(* Logix 5000 project; controller cal1632 1756-L62 rev 16.20; software revision 16.05; part 49 of 61 *)
(* tags used below, declared in another part *)
   FAULT : BOOL;
   HMI : BOOL;
   p01_recipe_active : recipe;
   p01r02 : routine;
   p01r09_pb_global_reset : BOOL;
   p27_ao_dia_a : REAL;
   p27_ao_dia_b : REAL;
   p27_inactive_tension_sp : REAL;
   p27r03_lower_A_tension_on : BOOL;
   p27r03_lower_B_tension_on : BOOL;
   p27r10 : routine;
   p27r10_lla_selected_tension : REAL;
   p27r10_llb_selected_tension : REAL;
   p27r10_timer_fault : TIMER[4];
   p27r10_timer_warning : TIMER[4];
   p27r10_unwind_a_brake_torque : REAL;
   p27r10_unwind_a_dia_ft : REAL;
   p27r10_unwind_b_brake_torque : REAL;
   p27r10_unwind_b_dia_ft : REAL;
   p28_ai_slitter_amps : REAL;
   p28_ai_slitter_hz : REAL;
   p28_ai_slitter_speed : REAL;
   p28_ao_sltr_selected_speed : REAL;
   p28_di_brake : BOOL;
   p28_di_motor : BOOL;
   p28_di_slitter : acs800_di_normal;
   p28_dint_to_hmi : DINT[16];
   p28_do_slt_air_supply_sv : BOOL;
   p28_do_sltr : acs800_do_normal;
   p28r01 : routine;
   p28r02 : routine;
   p28r02_fault_exists : BOOL;
   p28r02_timer_fault : TIMER[4];
   p28r02_timer_warning : TIMER[4];
   p28r02_unack_fault : BOOL;
   p28r02_unack_warning : BOOL;
   p28r02_warning_exists : BOOL;
   p28r03 : routine;
   p28r03_hz : SYS_SCP;
   p28r03_slitter_speed_fb : SYS_RPM_TO_SPEED;
   p28r03_timer_fault : TIMER[4];
   p28r03_timer_warning : TIMER[4];
   p28r04 : routine;
   p28r04_slitter_gear_ratio : REAL;
   p28r04_slitter_roll_diameter_ft : REAL;
   p28r04_slitter_speed : SYS_SPEED_TO_VFD;
   p28r04_timer_fault : TIMER[4];
   p28r04_timer_warning : TIMER[4];
   p28r05 : routine;
   p28r05_timer_fault : TIMER[4];
   p28r05_timer_warning : TIMER[4];
   p28r06 : routine;
   p28r07 : routine;
   p28r08 : routine;
   p28r09 : routine;
   p28r10_request_line_run : BOOL;
   p28r11 : routine;
   p28r11_slitter_on : BOOL;
(* P27_Lower_Poly_Letoff, continued *)

ROUTINE R10_Tension   (* ladder *)
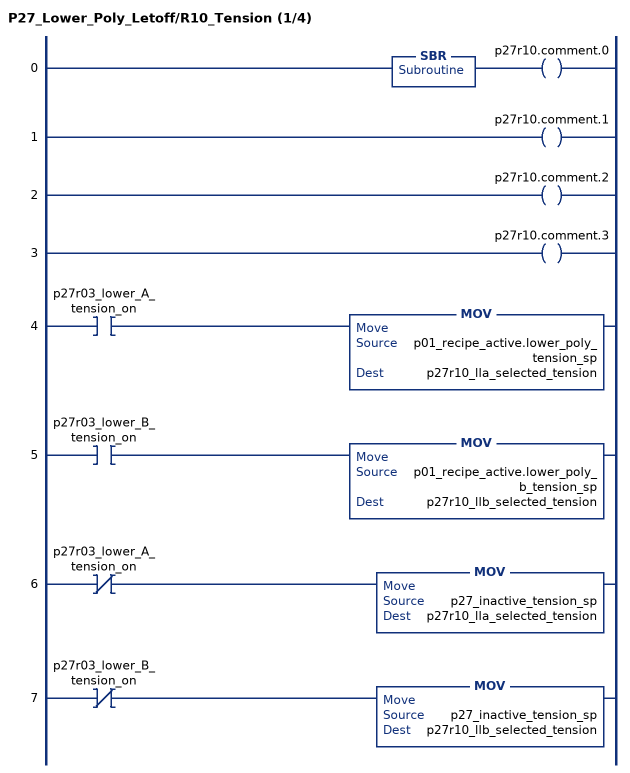
   0: SBR()OTE(p27r10.comment.0);
   1: OTE(p27r10.comment.1);
   2: OTE(p27r10.comment.2);
   3: OTE(p27r10.comment.3);
   4: XIC(p27r03_lower_A_tension_on)MOV(p01_recipe_active.lower_poly_tension_sp,p27r10_lla_selected_tension);
   5: XIC(p27r03_lower_B_tension_on)MOV(p01_recipe_active.lower_poly_b_tension_sp,p27r10_llb_selected_tension);
   6: XIO(p27r03_lower_A_tension_on)MOV(p27_inactive_tension_sp,p27r10_lla_selected_tension);
   7: XIO(p27r03_lower_B_tension_on)MOV(p27_inactive_tension_sp,p27r10_llb_selected_tension);
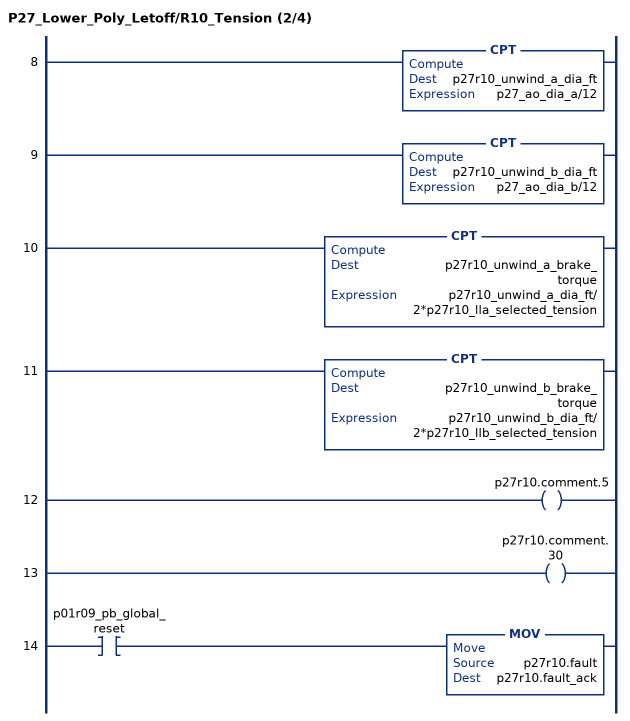
   8: CPT(p27r10_unwind_a_dia_ft,p27_ao_dia_a/12);
   9: CPT(p27r10_unwind_b_dia_ft,p27_ao_dia_b/12);
   10: CPT(p27r10_unwind_a_brake_torque,p27r10_unwind_a_dia_ft/2*p27r10_lla_selected_tension);
   11: CPT(p27r10_unwind_b_brake_torque,p27r10_unwind_b_dia_ft/2*p27r10_llb_selected_tension);
   12: OTE(p27r10.comment.5);
   13: OTE(p27r10.comment.30);
   14: XIC(p01r09_pb_global_reset)MOV(p27r10.fault,p27r10.fault_ack);
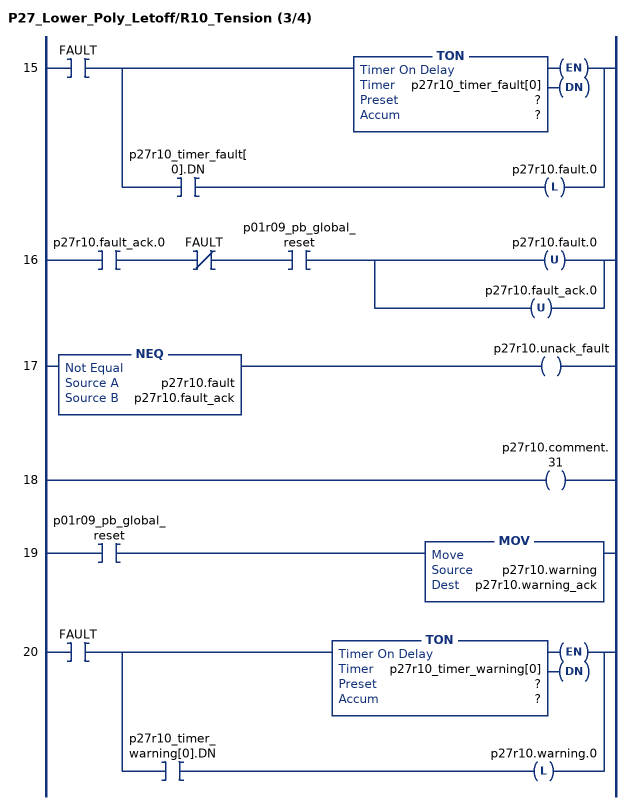
   15: XIC(FAULT)[TON(p27r10_timer_fault[0],?,?) ,XIC(p27r10_timer_fault[0].DN) OTL(p27r10.fault.0) ];
   16: XIC(p27r10.fault_ack.0)XIO(FAULT)XIC(p01r09_pb_global_reset)[OTU(p27r10.fault.0) ,OTU(p27r10.fault_ack.0) ];
   17: NEQ(p27r10.fault,p27r10.fault_ack)OTE(p27r10.unack_fault);
   18: OTE(p27r10.comment.31);
   19: XIC(p01r09_pb_global_reset)MOV(p27r10.warning,p27r10.warning_ack);
   20: XIC(FAULT)[TON(p27r10_timer_warning[0],?,?) ,XIC(p27r10_timer_warning[0].DN) OTL(p27r10.warning.0) ];
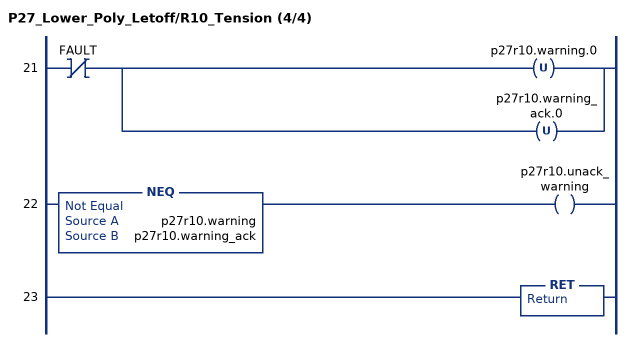
   21: XIO(FAULT)[OTU(p27r10.warning.0) ,OTU(p27r10.warning_ack.0) ];
   22: NEQ(p27r10.warning,p27r10.warning_ack)OTE(p27r10.unack_warning);
   23: RET();
END_ROUTINE
END_PROGRAM

PROGRAM P28_Slitter   (* main routine R01_Main *)

ROUTINE R01_Main   (* ladder *)
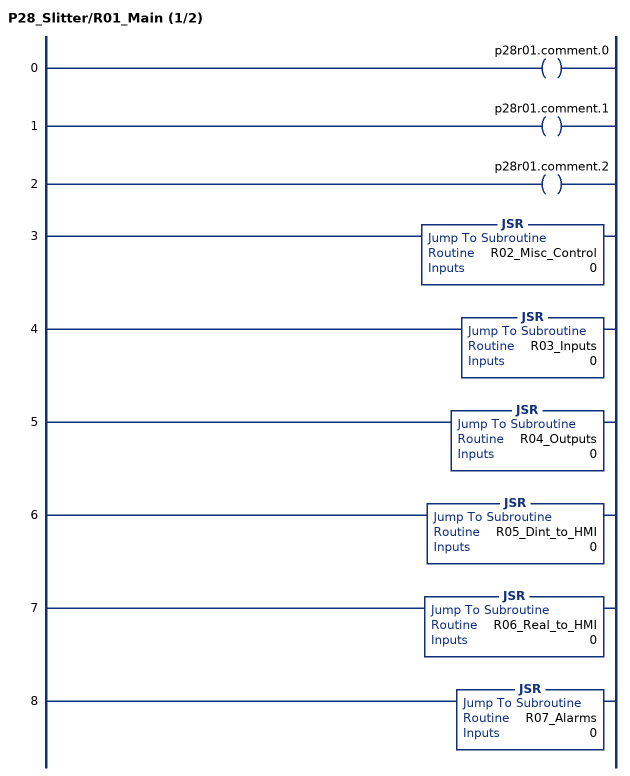
   0: OTE(p28r01.comment.0);
   1: OTE(p28r01.comment.1);
   2: OTE(p28r01.comment.2);
   3: JSR(R02_Misc_Control,0);
   4: JSR(R03_Inputs,0);
   5: JSR(R04_Outputs,0);
   6: JSR(R05_Dint_to_HMI,0);
   7: JSR(R06_Real_to_HMI,0);
   8: JSR(R07_Alarms,0);
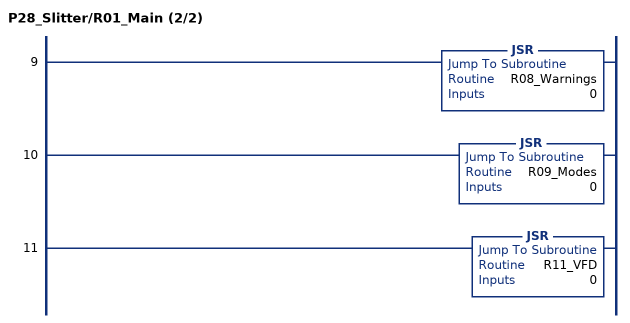
   9: JSR(R08_Warnings,0);
   10: JSR(R09_Modes,0);
   11: JSR(R11_VFD,0);
END_ROUTINE

ROUTINE R02_Misc_Control   (* ladder *)
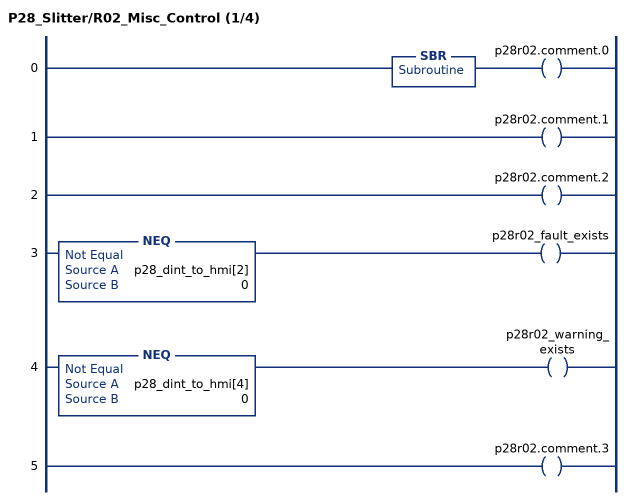
   0: SBR()OTE(p28r02.comment.0);
   1: OTE(p28r02.comment.1);
   2: OTE(p28r02.comment.2);
   3: NEQ(p28_dint_to_hmi[2],0)OTE(p28r02_fault_exists);
   4: NEQ(p28_dint_to_hmi[4],0)OTE(p28r02_warning_exists);
   5: OTE(p28r02.comment.3);
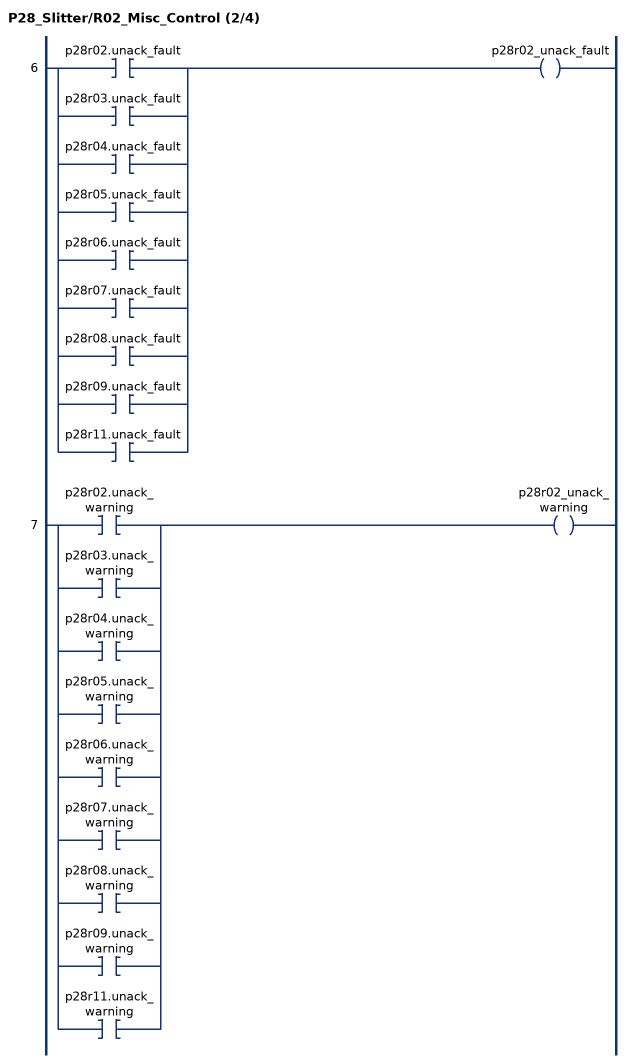
   6: [XIC(p28r02.unack_fault) ,XIC(p28r03.unack_fault) ,XIC(p28r04.unack_fault) ,XIC(p28r05.unack_fault) ,XIC(p28r06.unack_fault) ,XIC(p28r07.unack_fault) ,XIC(p28r08.unack_fault) ,XIC(p28r09.unack_fault) ,XIC(p28r11.unack_fault) ]OTE(p28r02_unack_fault);
   7: [XIC(p28r02.unack_warning) ,XIC(p28r03.unack_warning) ,XIC(p28r04.unack_warning) ,XIC(p28r05.unack_warning) ,XIC(p28r06.unack_warning) ,XIC(p28r07.unack_warning) ,XIC(p28r08.unack_warning) ,XIC(p28r09.unack_warning) ,XIC(p28r11.unack_warning) ]OTE(p28r02_unack_warning);
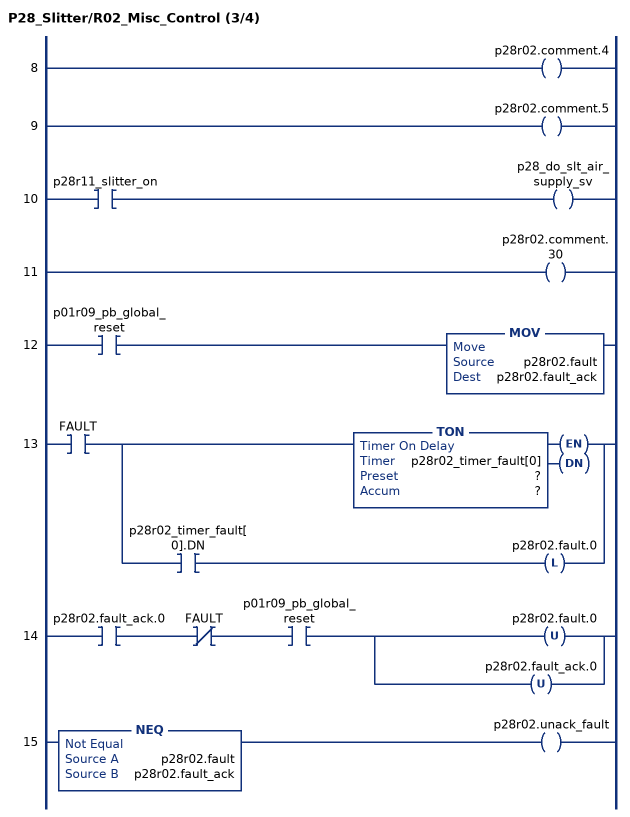
   8: OTE(p28r02.comment.4);
   9: OTE(p28r02.comment.5);
   10: XIC(p28r11_slitter_on)OTE(p28_do_slt_air_supply_sv);
   11: OTE(p28r02.comment.30);
   12: XIC(p01r09_pb_global_reset)MOV(p28r02.fault,p28r02.fault_ack);
   13: XIC(FAULT)[TON(p28r02_timer_fault[0],?,?) ,XIC(p28r02_timer_fault[0].DN) OTL(p28r02.fault.0) ];
   14: XIC(p28r02.fault_ack.0)XIO(FAULT)XIC(p01r09_pb_global_reset)[OTU(p28r02.fault.0) ,OTU(p28r02.fault_ack.0) ];
   15: NEQ(p28r02.fault,p28r02.fault_ack)OTE(p28r02.unack_fault);
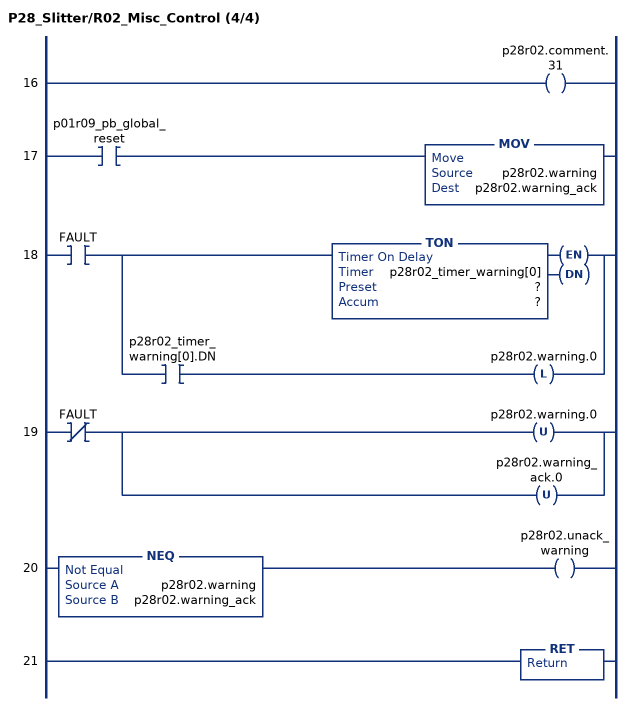
   16: OTE(p28r02.comment.31);
   17: XIC(p01r09_pb_global_reset)MOV(p28r02.warning,p28r02.warning_ack);
   18: XIC(FAULT)[TON(p28r02_timer_warning[0],?,?) ,XIC(p28r02_timer_warning[0].DN) OTL(p28r02.warning.0) ];
   19: XIO(FAULT)[OTU(p28r02.warning.0) ,OTU(p28r02.warning_ack.0) ];
   20: NEQ(p28r02.warning,p28r02.warning_ack)OTE(p28r02.unack_warning);
   21: RET();
END_ROUTINE

ROUTINE R03_Inputs   (* ladder *)
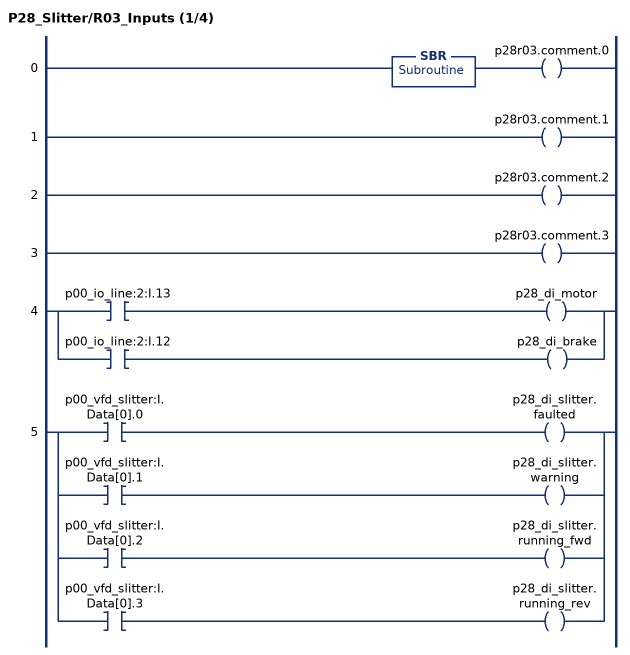
   0: SBR()OTE(p28r03.comment.0);
   1: OTE(p28r03.comment.1);
   2: OTE(p28r03.comment.2);
   3: OTE(p28r03.comment.3);
   4: [XIC(p00_io_line:2:I.13) OTE(p28_di_motor) ,XIC(p00_io_line:2:I.12) OTE(p28_di_brake) ];
   5: [XIC(p00_vfd_slitter:I.Data[0].0) OTE(p28_di_slitter.faulted) ,XIC(p00_vfd_slitter:I.Data[0].1) OTE(p28_di_slitter.warning) ,XIC(p00_vfd_slitter:I.Data[0].2) OTE(p28_di_slitter.running_fwd) ,XIC(p00_vfd_slitter:I.Data[0].3) OTE(p28_di_slitter.running_rev) ];
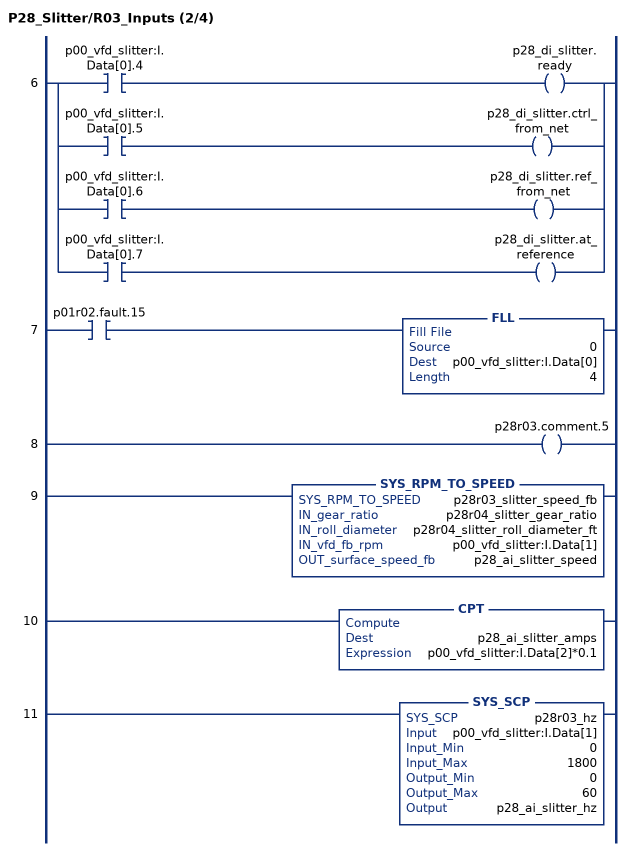
   6: [XIC(p00_vfd_slitter:I.Data[0].4) OTE(p28_di_slitter.ready) ,XIC(p00_vfd_slitter:I.Data[0].5) OTE(p28_di_slitter.ctrl_from_net) ,XIC(p00_vfd_slitter:I.Data[0].6) OTE(p28_di_slitter.ref_from_net) ,XIC(p00_vfd_slitter:I.Data[0].7) OTE(p28_di_slitter.at_reference) ];
   7: XIC(p01r02.fault.15)FLL(0,p00_vfd_slitter:I.Data[0],4);
   8: OTE(p28r03.comment.5);
   9: SYS_RPM_TO_SPEED(p28r03_slitter_speed_fb,p28r04_slitter_gear_ratio,p28r04_slitter_roll_diameter_ft,p00_vfd_slitter:I.Data[1],p28_ai_slitter_speed);
   10: CPT(p28_ai_slitter_amps,p00_vfd_slitter:I.Data[2]*0.1);
   11: SYS_SCP(p28r03_hz,p00_vfd_slitter:I.Data[1],0,1800,0,60,p28_ai_slitter_hz);
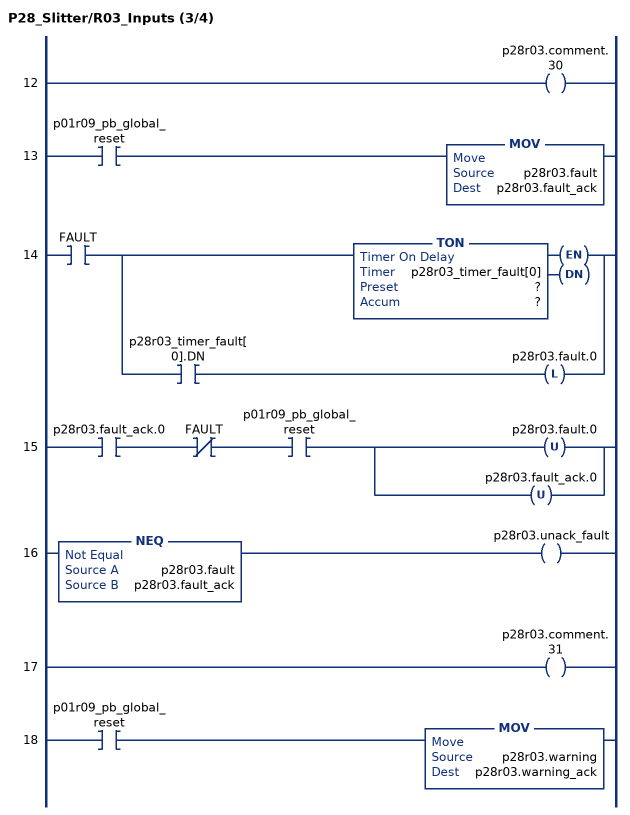
   12: OTE(p28r03.comment.30);
   13: XIC(p01r09_pb_global_reset)MOV(p28r03.fault,p28r03.fault_ack);
   14: XIC(FAULT)[TON(p28r03_timer_fault[0],?,?) ,XIC(p28r03_timer_fault[0].DN) OTL(p28r03.fault.0) ];
   15: XIC(p28r03.fault_ack.0)XIO(FAULT)XIC(p01r09_pb_global_reset)[OTU(p28r03.fault.0) ,OTU(p28r03.fault_ack.0) ];
   16: NEQ(p28r03.fault,p28r03.fault_ack)OTE(p28r03.unack_fault);
   17: OTE(p28r03.comment.31);
   18: XIC(p01r09_pb_global_reset)MOV(p28r03.warning,p28r03.warning_ack);
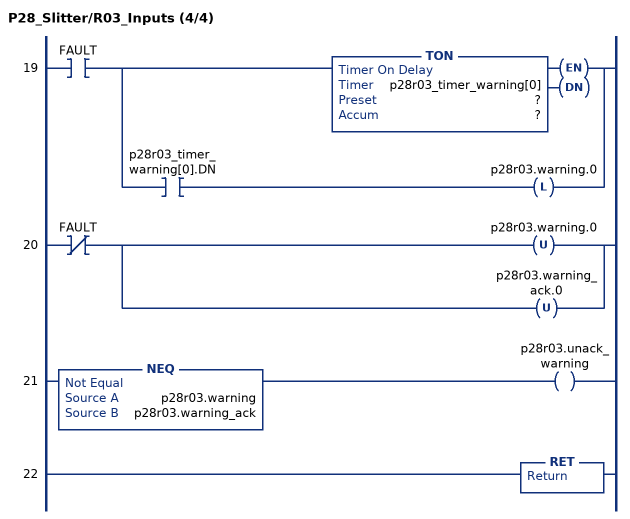
   19: XIC(FAULT)[TON(p28r03_timer_warning[0],?,?) ,XIC(p28r03_timer_warning[0].DN) OTL(p28r03.warning.0) ];
   20: XIO(FAULT)[OTU(p28r03.warning.0) ,OTU(p28r03.warning_ack.0) ];
   21: NEQ(p28r03.warning,p28r03.warning_ack)OTE(p28r03.unack_warning);
   22: RET();
END_ROUTINE

ROUTINE R04_Outputs   (* ladder *)
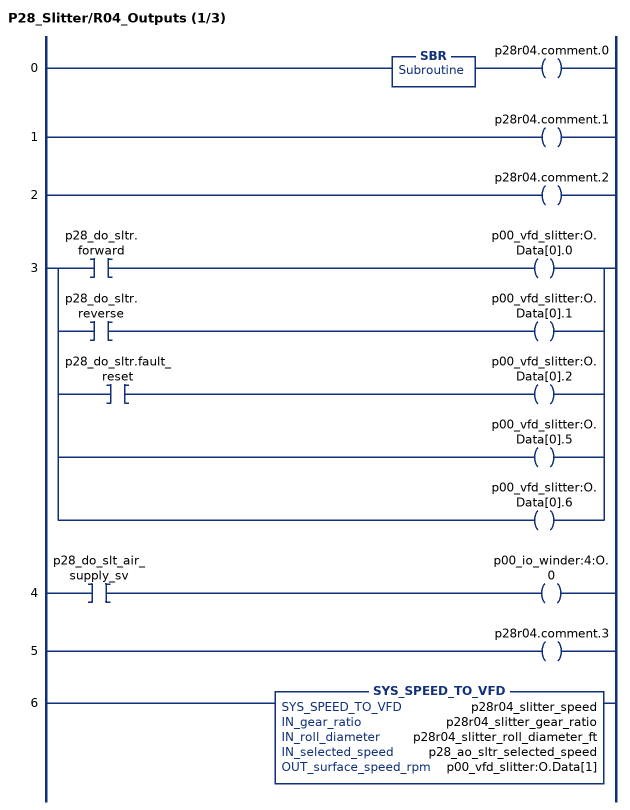
   0: SBR()OTE(p28r04.comment.0);
   1: OTE(p28r04.comment.1);
   2: OTE(p28r04.comment.2);
   3: [XIC(p28_do_sltr.forward) OTE(p00_vfd_slitter:O.Data[0].0) ,XIC(p28_do_sltr.reverse) OTE(p00_vfd_slitter:O.Data[0].1) ,XIC(p28_do_sltr.fault_reset) OTE(p00_vfd_slitter:O.Data[0].2) ,OTE(p00_vfd_slitter:O.Data[0].5) ,OTE(p00_vfd_slitter:O.Data[0].6) ];
   4: XIC(p28_do_slt_air_supply_sv)OTE(p00_io_winder:4:O.0);
   5: OTE(p28r04.comment.3);
   6: SYS_SPEED_TO_VFD(p28r04_slitter_speed,p28r04_slitter_gear_ratio,p28r04_slitter_roll_diameter_ft,p28_ao_sltr_selected_speed,p00_vfd_slitter:O.Data[1]);
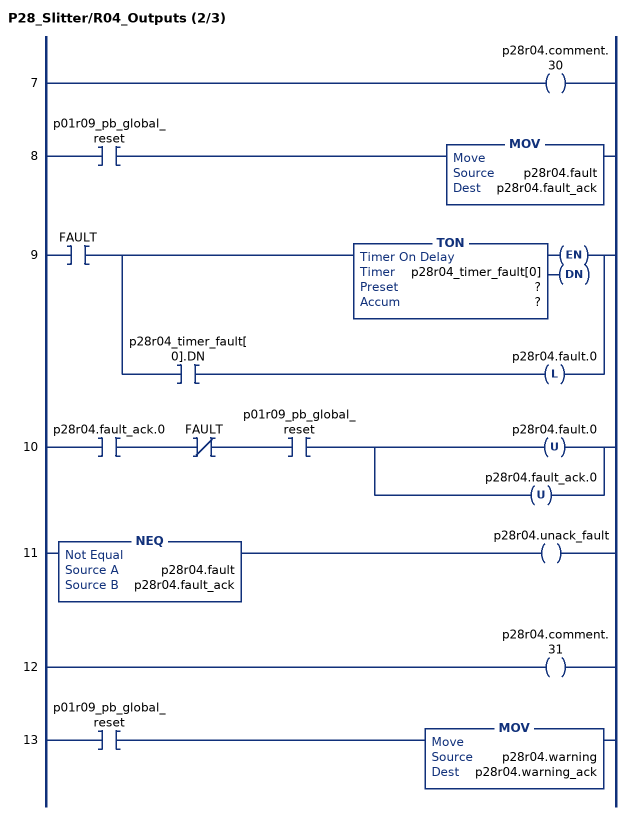
   7: OTE(p28r04.comment.30);
   8: XIC(p01r09_pb_global_reset)MOV(p28r04.fault,p28r04.fault_ack);
   9: XIC(FAULT)[TON(p28r04_timer_fault[0],?,?) ,XIC(p28r04_timer_fault[0].DN) OTL(p28r04.fault.0) ];
   10: XIC(p28r04.fault_ack.0)XIO(FAULT)XIC(p01r09_pb_global_reset)[OTU(p28r04.fault.0) ,OTU(p28r04.fault_ack.0) ];
   11: NEQ(p28r04.fault,p28r04.fault_ack)OTE(p28r04.unack_fault);
   12: OTE(p28r04.comment.31);
   13: XIC(p01r09_pb_global_reset)MOV(p28r04.warning,p28r04.warning_ack);
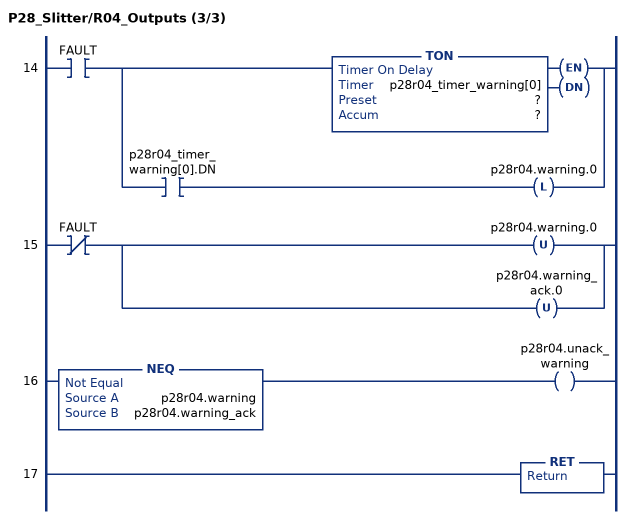
   14: XIC(FAULT)[TON(p28r04_timer_warning[0],?,?) ,XIC(p28r04_timer_warning[0].DN) OTL(p28r04.warning.0) ];
   15: XIO(FAULT)[OTU(p28r04.warning.0) ,OTU(p28r04.warning_ack.0) ];
   16: NEQ(p28r04.warning,p28r04.warning_ack)OTE(p28r04.unack_warning);
   17: RET();
END_ROUTINE

ROUTINE R05_Dint_to_HMI   (* ladder *)
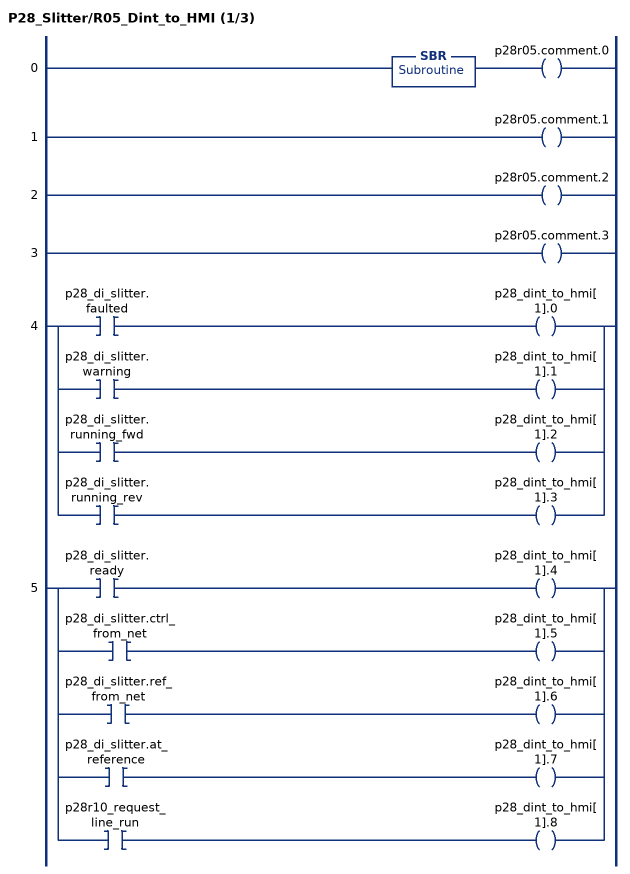
   0: SBR()OTE(p28r05.comment.0);
   1: OTE(p28r05.comment.1);
   2: OTE(p28r05.comment.2);
   3: OTE(p28r05.comment.3);
   4: [XIC(p28_di_slitter.faulted) OTE(p28_dint_to_hmi[1].0) ,XIC(p28_di_slitter.warning) OTE(p28_dint_to_hmi[1].1) ,XIC(p28_di_slitter.running_fwd) OTE(p28_dint_to_hmi[1].2) ,XIC(p28_di_slitter.running_rev) OTE(p28_dint_to_hmi[1].3) ];
   5: [XIC(p28_di_slitter.ready) OTE(p28_dint_to_hmi[1].4) ,XIC(p28_di_slitter.ctrl_from_net) OTE(p28_dint_to_hmi[1].5) ,XIC(p28_di_slitter.ref_from_net) OTE(p28_dint_to_hmi[1].6) ,XIC(p28_di_slitter.at_reference) OTE(p28_dint_to_hmi[1].7) ,XIC(p28r10_request_line_run) OTE(p28_dint_to_hmi[1].8) ];
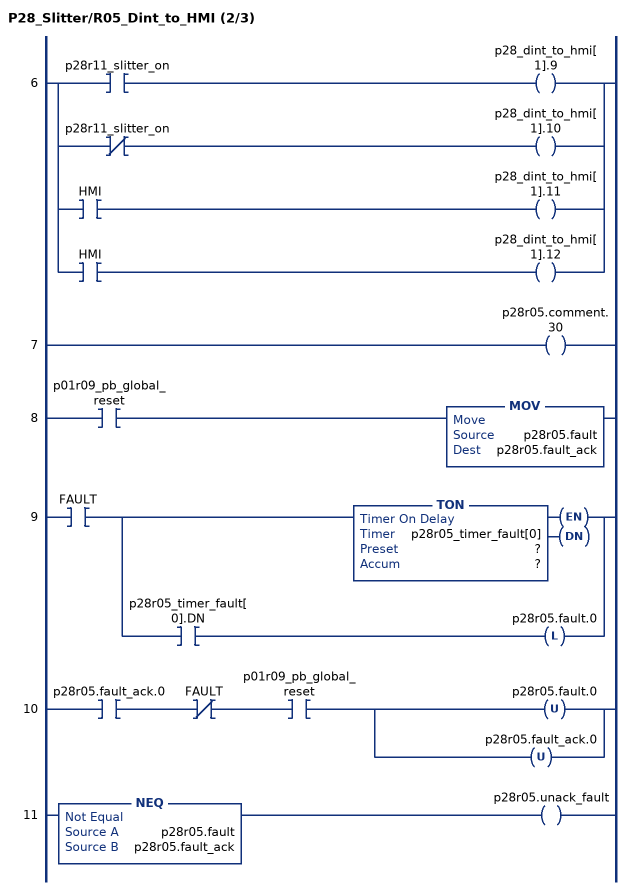
   6: [XIC(p28r11_slitter_on) OTE(p28_dint_to_hmi[1].9) ,XIO(p28r11_slitter_on) OTE(p28_dint_to_hmi[1].10) ,XIC(HMI) OTE(p28_dint_to_hmi[1].11) ,XIC(HMI) OTE(p28_dint_to_hmi[1].12) ];
   7: OTE(p28r05.comment.30);
   8: XIC(p01r09_pb_global_reset)MOV(p28r05.fault,p28r05.fault_ack);
   9: XIC(FAULT)[TON(p28r05_timer_fault[0],?,?) ,XIC(p28r05_timer_fault[0].DN) OTL(p28r05.fault.0) ];
   10: XIC(p28r05.fault_ack.0)XIO(FAULT)XIC(p01r09_pb_global_reset)[OTU(p28r05.fault.0) ,OTU(p28r05.fault_ack.0) ];
   11: NEQ(p28r05.fault,p28r05.fault_ack)OTE(p28r05.unack_fault);
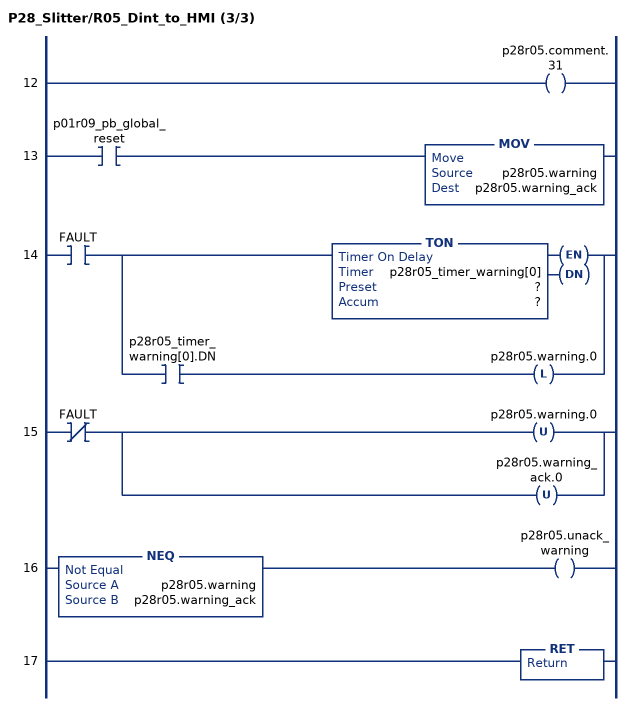
   12: OTE(p28r05.comment.31);
   13: XIC(p01r09_pb_global_reset)MOV(p28r05.warning,p28r05.warning_ack);
   14: XIC(FAULT)[TON(p28r05_timer_warning[0],?,?) ,XIC(p28r05_timer_warning[0].DN) OTL(p28r05.warning.0) ];
   15: XIO(FAULT)[OTU(p28r05.warning.0) ,OTU(p28r05.warning_ack.0) ];
   16: NEQ(p28r05.warning,p28r05.warning_ack)OTE(p28r05.unack_warning);
   17: RET();
END_ROUTINE
